Universal Robots PolyScope program: AlvarezZavaleta_LuisAlberto_P1.urp

Program First1 (installation=default directory=/home/ur/ursim-current/programs createdIn=5.14.5 lastSavedIn=5.14.5 robotSerialNumber=20195399999)
Calibrated DH parameters: a=[0, -0.24355, -0.2132, 0, 0, 0]; d=[0.15185, 0, 0, 0.13105, 0.08535, 0.0921]; alpha=[1.570796, 0, 0, 1.570796, -1.570796, 0]; deltaTheta=[0, 0, 0, 0, 0, 0]
InitVariablesNode
Robot Program (runOnlyOnce=true)
  MoveL speed 250 mm/s, acceleration 1200 mm/s^2 (useActiveTCP=true) feature=Base
    Waypoint Inicial: TCP in base x=-136.862 y=-267.181 z=146.98 mm, rx=-0.0012 ry=3.1163 rz=0.0389 rad; joints [-91.713, -98.954, -126.222, -46.298, 91.392, -1.776] deg
    MoveDirectionNode expression=[-0.25,0,0.75]; feature=Joint_6_name
      Until DISTANCE (allowActions=false deceleration=3 distanceNodeType=STOP) Distance=0.11; motionParameters(blendRadius=0)
    MoveDirectionNode (selectedDirection=XPlus) feature=Joint_6_name
      Until DISTANCE (allowActions=false deceleration=3 distanceNodeType=STOP) Distance=0.07; motionParameters(blendRadius=0)
    Waypoint Inicial: TCP in base x=-136.862 y=-267.181 z=146.98 mm, rx=-0.0012 ry=3.1163 rz=0.0389 rad; joints [-91.713, -98.954, -126.222, -46.298, 91.392, -1.776] deg
